% RSLogix 500 project I2P Job 11 - Myah.RSS, saved by version 10.00.00.00 %
PROJECT "ML05B"    % processor: Bul.1763 MicroLogix 1100 Series B %

PROGRAM FILES
  LAD 2   8 rungs

DATA FILES
  O0 OUTPUT  4 elements
  I1 INPUT  6 elements
  S2 STATUS  66 elements
  B3 BINARY  1 elements
  T4 TIMER  1 elements
  C5 COUNTER  1 elements
  R6 CONTROL  1 elements
  N7 INTEGER  1 elements
  F8 FLOAT  1 elements

LADDER 2
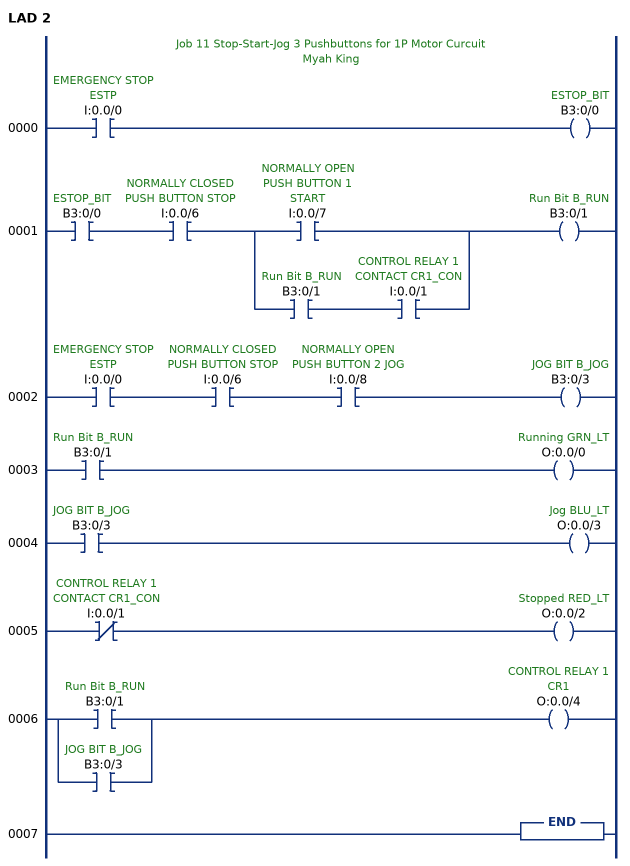
% Rung: 0 %
% Job 11 Stop-Start-Jog 3 Pushbuttons for 1P Motor Curcuit
% Myah King %
SOR XIC I:0.0/0 OTE B3:0/0 EOR
%   I:0.0/0  ESTP  "EMERGENCY STOP" %
%   B3:0/0  ESTOP_BIT %
% Rung: 1 %
SOR XIC B3:0/0 XIC I:0.0/6 BST XIC I:0.0/7 NXB XIC B3:0/1 XIC I:0.0/1 BND OTE B3:0/1 EOR
%   B3:0/0  ESTOP_BIT %
%   I:0.0/6  STOP  "NORMALLY CLOSED PUSH BUTTON" %
%   I:0.0/7  START  "NORMALLY OPEN PUSH BUTTON 1" %
%   B3:0/1  B_RUN  "Run Bit" %
%   I:0.0/1  CR1_CON  "CONTROL RELAY 1 CONTACT" %
% Rung: 2 %
SOR XIC I:0.0/0 XIC I:0.0/6 XIC I:0.0/8 OTE B3:0/3 EOR
%   I:0.0/0  ESTP  "EMERGENCY STOP" %
%   I:0.0/6  STOP  "NORMALLY CLOSED PUSH BUTTON" %
%   I:0.0/8  JOG  "NORMALLY OPEN PUSH BUTTON 2" %
%   B3:0/3  B_JOG  "JOG BIT" %
% Rung: 3 %
SOR XIC B3:0/1 OTE O:0.0/0 EOR
%   B3:0/1  B_RUN  "Run Bit" %
%   O:0.0/0  GRN_LT  "Running" %
% Rung: 4 %
SOR XIC B3:0/3 OTE O:0.0/3 EOR
%   B3:0/3  B_JOG  "JOG BIT" %
%   O:0.0/3  BLU_LT  "Jog" %
% Rung: 5 %
SOR XIO I:0.0/1 OTE O:0.0/2 EOR
%   I:0.0/1  CR1_CON  "CONTROL RELAY 1 CONTACT" %
%   O:0.0/2  RED_LT  "Stopped" %
% Rung: 6 %
SOR BST XIC B3:0/1 NXB XIC B3:0/3 BND OTE O:0.0/4 EOR
%   B3:0/1  B_RUN  "Run Bit" %
%   B3:0/3  B_JOG  "JOG BIT" %
%   O:0.0/4  CR1  "CONTROL RELAY 1" %
% Rung: 7 %
SOR END EOR

OTHER DOCUMENTED ADDRESSES
  I:0.0/2  CR2_CON  "CONTROL RELAY 2 CON"
  I:0.0/3  3PSS_A  "3 POSITION SELCTOR SWITCH A POSITION"
  I:0.0/4  3PSS_B  "3 POSITION SELECTOR SWITCH B POSITON"
  I:0.0/5  2PSS  "2 POSITION SELECTOR SWITCH"
  O:0.0/1  YLW_LT  "YELLOW LIGHT"
  O:0.0/5  CR2  "CONTROL RELAY 2"

DATA TABLE (non-zero values as saved)
DATA B3
% B3:0 % 0X0001
